TYPE stISS :
STRUCT
	//R//						
		error_code			:INT;
		state						:INT;
		mainTankLevel		:LREAL;
		Init_Done				:BOOL;
		Error						:BOOL;
	//W//
		Initialize				:BOOL;	//  
		Setoff				:BOOL;	//  
		sensor_blink		:BOOL;
END_STRUCT
END_TYPE

(* stored: Version 1.1.0.1, ProductVersion 3.1.4024.11
   DUT stISS: Id {c3abb084-1816-46cf-b1c3-03e028401aff} *)
